FUNCTION_BLOCK SBT IMPLEMENTS MachineModule
VAR
	bEnable			: BOOL;
	bDisable        : BOOL;
	bError          : BOOL;
	bOverride       : BOOL;
	bSimulation     : BOOL;
	bStart          : BOOL;
	bStop           : BOOL;
END_VAR

// This is the core module needed that we are creating for our STS and contains everything related to the STS

// To be added
(*
FEEDER

SAT

VBT

EJECT

GATE

SBT

*)

METHOD Disable : BOOL
VAR_INPUT
END_VAR
bEnable:=FALSE;
END_METHOD

METHOD Enable : BOOL
VAR_INPUT
END_VAR
bEnable:=TRUE;
bDisable:=False;
END_METHOD

METHOD Error : BOOL
VAR_INPUT
END_VAR
bEnable:=FALSE;
END_METHOD

METHOD Override : BOOL
VAR_INPUT
END_VAR
END_METHOD

METHOD Reset : BOOL
VAR_INPUT
END_VAR
END_METHOD

METHOD Start : BOOL
VAR_INPUT
END_VAR
END_METHOD

METHOD PUBLIC StateMachine
VAR_INPUT
END_VAR
END_METHOD

METHOD Stop : BOOL
VAR_INPUT
END_VAR
END_METHOD

END_FUNCTION_BLOCK

(* stored: Version 1.1.0.1, ProductVersion 3.1.4024.12
   POU SBT: Id {a1135cdb-167b-4fe2-8ee0-f9a094475996}, SpecialFunc None
   Method Disable: Id {a85da843-6af5-4c59-9648-6b66c1a39a28}
   Method Enable: Id {803ba3ae-99bc-44de-8d22-6c03af03061b}
   Method Error: Id {ac5ae575-af06-444c-84ea-84013cff3df0}
   Method Override: Id {169ffa85-df2c-4b2e-a466-3e052ab788bd}
   Method Reset: Id {3b6b125f-3337-4662-bcfd-2dd9ce78e7f0}
   Method Start: Id {ec57ec5a-7fc3-48d8-ae55-9cd26dae6ba1}
   Method StateMachine: Id {356580bc-9cc1-4ae7-aeda-0340140a8b43}
   Method Stop: Id {adfbd9b0-30a5-4f90-a0b5-477935bf1b6d} *)
